# EPICS substitutions: ek9000App/Db/EL1014_mbbiDirect.substitutions
file EL1014.template
{       pattern
        {
                TERMINAL,

        }
        {
        }
}
